FUNCTION Convert_LINT_TO_DT : Hresult
VAR_INPUT
	in : LINT;
	out : REFERENCE TO DT;
END_VAR
VAR
	converted : DT;
END_VAR

converted := LINT_TO_DT(in);

IF (DT_TO_LINT(converted) <> in) THEN
	Convert_LINT_TO_DT := INCOMPATIBLE;
	RETURN;
END_IF

out := converted;

END_FUNCTION

(* stored: Version 1.1.0.1, ProductVersion 3.1.4024.12
   POU Convert_LINT_TO_DT: Id {7e9b2819-886a-4609-aec9-02b40523826a}, SpecialFunc None *)
